TYPE Read_BLVac1_Values_To_PC_Struct :
UNION
	S_BLVac1Values_To_PC:S_BLVac1Values_To_PC_Struct;
END_UNION
END_TYPE

(* stored: Version 1.1.0.1, ProductVersion 3.1.4024.16
   DUT Read_BLVac1_Values_To_PC_Struct: Id {f74278db-a8f0-4e3a-b478-e56b980e48f7} *)
